FUNCTION_BLOCK FB_StateError IMPLEMENTS I_State
VAR
	_refMainStateMachine		: REFERENCE TO FB_MainStateMachine;
	_fbXmlSrvRead				: FB_XmlSrvRead;
	_nErrorAckCount				: UDINT;
END_VAR

METHOD FB_init : BOOL
VAR_INPUT
	// if TRUE, the retain variables are initialized (warm start / cold start)
	bInitRetains			: BOOL;
	// if TRUE, the instance afterwards gets moved into the copy code (online
	// change)
	bInCopyCode				: BOOL;
	fbMainStateMachine		: REFERENCE TO FB_MainStateMachine;
END_VAR
_refMainStateMachine REF= fbMainStateMachine;
END_METHOD

METHOD StopButtonPressed
END_METHOD

METHOD Execute
END_METHOD

METHOD SafetyTripped
END_METHOD

METHOD ClearErrors
END_METHOD

METHOD SafetyAcknowledged
END_METHOD

METHOD GetDescription : STRING
GetDescription := 'Error';
END_METHOD

METHOD StartButtonPressed
IF _refMainStateMachine.ipPrevState <> 0 THEN
	_nErrorAckCount := _nErrorAckCount + 1;
	_refMainStateMachine.ipPrevState.ClearErrors();
	_refMainStateMachine.SetState(_refMainStateMachine.ipPrevState);
END_IF
END_METHOD

END_FUNCTION_BLOCK

(* stored: Version 1.1.0.1, ProductVersion 3.1.4024.11
   POU FB_StateError: Id {eeed6ac7-e68c-4278-9d61-2c19f6c85117}, SpecialFunc None
   Method FB_init: Id {55065133-d105-4658-99bc-7a60d238c930}
   Method StopButtonPressed: Id {708b4350-9d95-4587-8c34-e780bb234fa2}
   Method Execute: Id {8737d1c4-23d2-4d12-a1c6-68dcd451482b}
   Method SafetyTripped: Id {95208b12-2d2c-4151-8da1-d5dd8514cbae}
   Method ClearErrors: Id {9fbd23a6-d862-486b-8486-4990db5535cc}
   Method SafetyAcknowledged: Id {b09610c4-425f-4b11-bb73-8e8af849c769}
   Method GetDescription: Id {c558a173-9014-4b09-9d2a-6eb6d4f7b8cc}
   Method StartButtonPressed: Id {d2b9d275-72b1-43b7-bc0b-ade5c7e5f2e1} *)
